PROGRAM MAIN
VAR
END_VAR

END_PROGRAM

(* stored: Version 1.1.0.1
   POU MAIN: Id {c9b6e0a8-4ace-475c-908a-3b86f1d3cf42} *)
